RoboDK station: Test-Universal_Robots.rdk

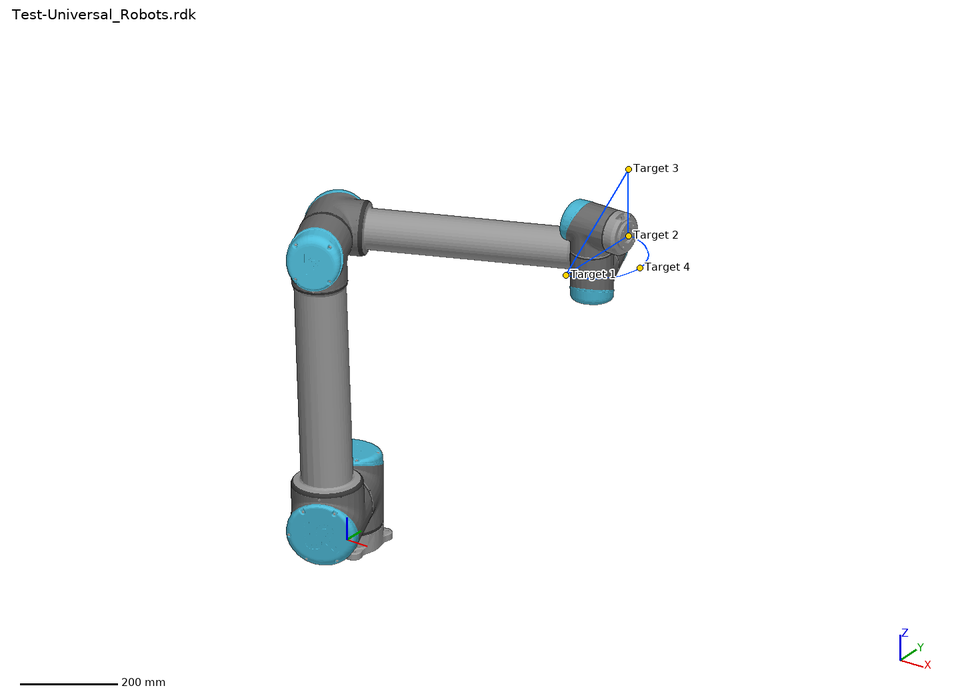
[picture v0: the station drawn from its stored meshes, robots at their saved joint values, targets as dots, program paths as lines]
Station Test-Universal-RObots. Poses are relative to the parent item; angles as X-Y-Z fixed-axis rotations.
Station parameters (name, value as stored): IO_5, 1
  - frame UR10 Base at (0, 0, 0) mm
    - robot UR10: 6 axes, payload 10 kg, reach 1300 mm, repeatability 0.1 mm, weight 28.9 kg
        modified DH rows (alpha deg, a mm, theta deg, d mm): 0, 0, 0, 128; 90, 0, 180, 0; 0, 612.7, 0, 0; 0, 571.6, 0, 163.9; -90, 0, 0, 115.7; 90, 0, 180, 92.2
        joint limits [-360, -360, -360, -360, -360, -360] to [360, 360, 360, 360, 360, 360]; home [0, -90, -90, 0, 90, 0]; saved at [22.599, -88.066, -91.899, -0.035, 67.401, 0]
    - target Target 1 (Cartesian target) at (663.8, -163.9, 856.4) mm, rotated rx -90 ry 0 rz -90 deg; joints [0, -90, -90, 0, 90, 0] of UR10
    - target Target 2 (Cartesian target) at (663.8, 60.39, 856.4) mm, rotated rx -90 ry 0 rz -90 deg; joints [22.599, -88.066, -91.899, -0.035, 67.401, 0] of UR10
    - target Target 3 (Cartesian target) at (663.8, 60.39, 1007.85) mm, rotated rx -90 ry 0 rz -90 deg; joints [22.599, -89.976, -74.66, -15.364, 67.401, 0] of UR10
    - target Target 4 (Cartesian target) at (768.37, -48.53, 856.4) mm, rotated rx -90 ry 0 rz -90 deg; joints [9.886, -98.09, -81.299, -0.611, 80.114, 0] of UR10
  - program Prog1 (13 instructions, listed below)
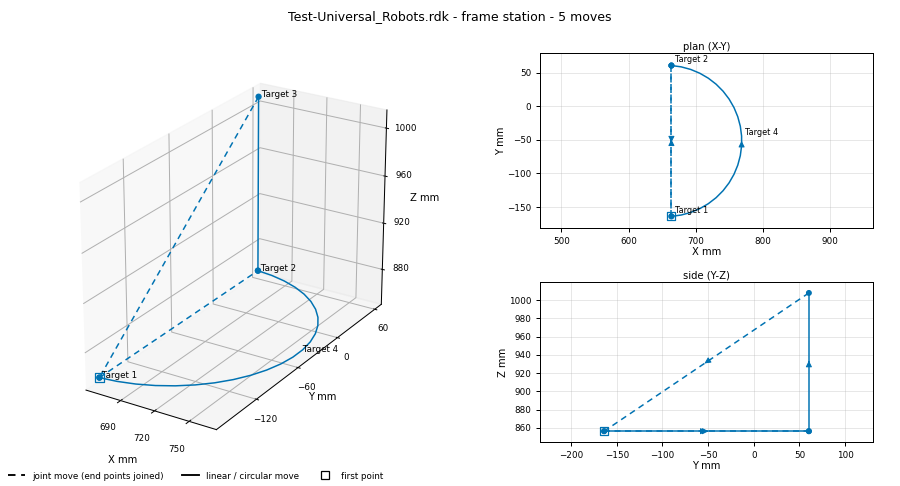
[picture p0: tool path of Test-Universal_Robots.rdk in frame station, 5 of 5 moves have a stored position in this frame; points joined in program order, loops and branches not executed]

--- program Prog1 (robot UR10) ---
  Set Ref.: UR10 Base
  MoveJ (Target 1)
  MoveJ (Target 2)
  MoveL (Target 3)
  MoveJ (Target 1)
  MoveC (Target 4, Target 2)
  Set speed (500.0 mm/s)
  Print: Display message
  Pause 500 ms
  Set IO_5=1
  Wait IO_5=1 T5.0s
  Set Ref.: UR10 Base
  Set Tool at (0, 0, 0) mm
